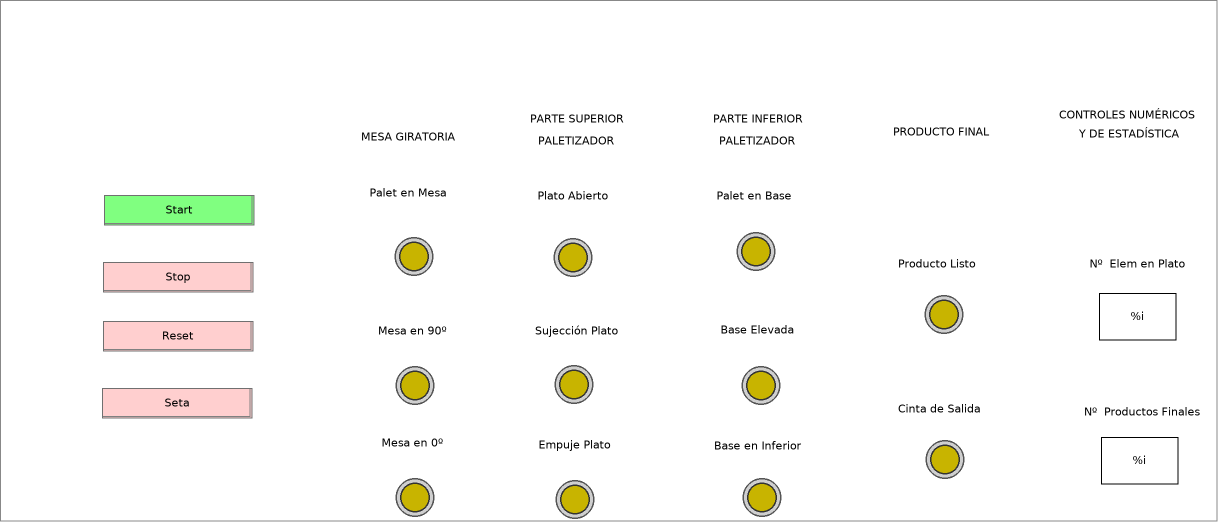
VISUALIZATION HMI  // 1218x522
    Button (104,195 150x30), "Start"
        toggle GVLvars.botonStart
    Button (103,262 150x30), "Stop", colour toggle: NOT GVLvars.botonStop
        toggle GVLvars.botonStop
    Button (103,321 150x30), "Reset", colour toggle: GVLvars.botonReset and MAIN.emergencia
        toggle GVLvars.botonReset
    Button (102,388 150x30), "Seta", colour toggle: Not GVLvars.seta
        toggle GVLvars.seta
    Lamp1 (918,292 52x45), variable: MAIN.paletizadoListo, style: Lamp-Lamp1-Yellow
    Label (890,249 97x30), "Producto Listo"
    Lamp1 (388,234 52x45), tooltip "Indicador de un palet sobre la mesa giratoria", variable: GVLvars.frontLimit, style: Lamp-Lamp1-Yellow
    Label (333,122 150x30), "MESA GIRATORIA"
    Lamp1 (389,363 52x45), tooltip "Indicador de mesa giratoria orientada a 90º", variable: GVLvars.maximunRotation, style: Lamp-Lamp1-Yellow
    Label (371,316 83x30), "Mesa en 90º"
    Label (650,185 190x42)
    Lamp1 (547,235 52x45), tooltip "Cinta con las bases y posteriormente producto final", variable: GVLvars.OpenPlate, style: Lamp-Lamp1-Yellow
    Label (519,175 108x42), "Plato Abierto"
    Lamp1 (548,362 52x45), tooltip "Cinta con las bases y posteriormente producto final", variable: GVLvars.moveClamper, style: Lamp-Lamp1-Yellow
    Label (519,310 115x42), "Sujección Plato"
    Label (333,178 150x30), "Palet en Mesa"
    Lamp1 (389,475 52x45), tooltip "Indicador de mesa giratoria orinetada a 0ª (posicion de reposo)", variable: GVLvars.minuminRotation, style: Lamp-Lamp1-Yellow
    Label (371,428 83x30), "Mesa en 0º"
    Label (502,104 150x30), "PARTE SUPERIOR"
    Label (501,126 150x30), "PALETIZADOR"
    Lamp1 (549,477 52x45), tooltip "Cinta con las bases y posteriormente producto final", variable: GVLvars.pusher, style: Lamp-Lamp1-Yellow
    Label (517,424 115x42), "Empuje Plato"
    Lamp1 (730,229 52x45), tooltip "Cinta con las bases y posteriormente producto final", variable: GVLvars.elevatorFrontLimit, style: Lamp-Lamp1-Yellow
    Label (700,175 108x42), "Palet en Base"
    Lamp1 (735,363 52x45), tooltip "Cinta con las bases y posteriormente producto final", variable: GVLvars.elevatorUp, style: Lamp-Lamp1-Yellow
    Label (700,309 115x42), "Base Elevada"
    Label (683,104 150x30), "PARTE INFERIOR"
    Label (682,126 150x30), "PALETIZADOR"
    Lamp1 (736,475 52x45), tooltip "Cinta con las bases y posteriormente producto final", variable: GVLvars.elevatorDown, style: Lamp-Lamp1-Yellow
    Label (700,425 115x42), "Base en Inferior"
    Label (1036,100 182x30), "CONTROLES NUMÉRICOS"
    Label (1056,119 150x30), "Y DE ESTADÍSTICA"
    Label (866,117 150x30), "PRODUCTO FINAL"
    Lamp1 (919,437 52x45), variable: GVLvars.cintaSalida, style: Lamp-Lamp1-Yellow
    Label (891,394 97x30), "Cinta de Salida"
    Rectangle (1099,293 77x47), "%i", tooltip "Indicador numérico de los elementos que se encuentran sobre el plato del paletizador", text variable: MAIN.contadorVector
    Label (1089,247 97x34), "Nº Elem en Plato"
    Rectangle (1101,437 77x47), "%i", tooltip "Indicador numérico de los elementos que se encuentran sobre el plato del paletizador", text variable: GVLvars.numProductosCompletos
    Label (1076,395 132x34), "Nº Productos Finales"
END_VISUALIZATION

(* stored: Version 1.1.0.1, ProductVersion 3.1.4024.15
   Visu HMI: Id {0d01b5ef-06f2-4d3d-9bea-c974f2ffaa85} *)
